VAR_GLOBAL
	SystemStarted		: BOOL;
	FlashBit			: BOOL;
	TransferBusy		: BOOL;
	TransferringLeft	: BOOL;
	TransferringRight	: BOOL;
	EmergencyActivated	: BOOL;
	BoxCounted			: WORD;
END_VAR

(* stored: Version 1.1.0.1, ProductVersion 3.1.4024.6
   GVL GeneralTags: Id {c2400427-fd7e-4217-8e00-2f0a56b4dc4b} *)
